TYPE DUT_1 :
STRUCT
END_STRUCT
END_TYPE

(* stored: Version 1.1.0.1, ProductVersion 3.1.4024.12
   DUT DUT_1: Id {7f5e4b18-1bfd-487f-a87f-f9689a5bad7a} *)
